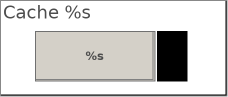
VISUALIZATION SA_CACHE_ACTUATOR2  // 228x97
VAR_IN_OUT
	m_Input_PRM_Forcage : Bool;
END_VAR
VAR_INPUT
	m_Input_CACHE : BLOCK_ACTUATOR2;
END_VAR
    RoundedRectangle (0,0 226x95), "Cache %s", text variable: m_Input_CACHE.MNEMO
    RoundedRectangle (157,31 30x50), colour toggle: m_Input_CACHE.STATE_ON
    Button (35,31 120x50), "%s", input disabled if: NOT (PRG_User.ACTU_USER.FONCTION_SA AND NOT MACHINE.STATE_PROD), text list: 'TextList_Orders', text index: 0
        toggle m_Input_PRM_Forcage
END_VISUALIZATION

(* stored: Version 1.1.0.1, ProductVersion 3.1.4024.10
   Visu SA_CACHE_ACTUATOR2: Id {1090dae1-1e70-4519-b55f-7b247fe13828} *)
